(* PLC project Tc2_SUPS.FB_S_UPS_CX9020_U900 Demo, tc3-libraries-kb TwinCAT 3.1 *)
(* stored: creationDateTime 2026-05-10T09:00:00, modificationDateTime 2026-05-10T09:00:00 *)

PROGRAM P_Demo_FB_S_UPS_CX9020_U900
  VAR
    fbFB_S_UPS_CX9020_U900 : FB_S_UPS_CX9020_U900;  (* CX9020-U900 实例 *)
    arg_sNetID : T_AmsNetId;  (* VAR_INPUT sNetID: 控制器 AmsNetId（空字符串表本地） *)
    arg_iPLCPort : UINT;  (* VAR_INPUT iPLCPort: 写持久化数据的 PLC runtime 端口（851/852/...，0 = 自动） *)
    arg_tTimeout : TIME;  (* VAR_INPUT tTimeout: ADS 超时（默认 DEFAULT_ADS_TIMEOUT） *)
    arg_eUpsMode : E_S_UPS_Mode;  (* VAR_INPUT eUpsMode: UPS 工作模式（默认 eSUPS_WrPersistData_Shutdown） *)
    arg_ePersistentMode : E_PersistentMode;  (* VAR_INPUT ePersistentMode: 持久化数据写入模式（默认 SPDM_2PASS） *)
    arg_tRecoverTime : TIME;  (* VAR_INPUT tRecoverTime: 短时断电恢复时间（默认 T#10s） *)
    out_bPowerFailDetect : BOOL;  (* VAR_OUTPUT bPowerFailDetect: 断电期间为 TRUE *)
    out_eState : E_S_UPS_State;  (* VAR_OUTPUT eState: FB 内部状态 *)
  END_VAR

            // ============================================================
// Tc2_SUPS.FB_S_UPS_CX9020_U900 演示程序
// ============================================================
// 场景：在 CX9020-U900 平台上接管 1-second UPS：检测断电时保存持久数据并执行 quick shutdown
// 验证步骤：
//   1. 引用 Tc2_SUPS（及其依赖：Tc2_System 等）
//   2. 编译 + 登录
//   3. 在线监视各 out_* 输出
//   4. 必要时按场景给 arg_* 输入赋值（详见 doc.md 的'使用注意'）
// ============================================================

fbFB_S_UPS_CX9020_U900(
    sNetID := arg_sNetID,
    iPLCPort := arg_iPLCPort,
    tTimeout := arg_tTimeout,
    eUpsMode := arg_eUpsMode,
    ePersistentMode := arg_ePersistentMode,
    tRecoverTime := arg_tRecoverTime,
    bPowerFailDetect => out_bPowerFailDetect,
    eState => out_eState
);

          
END_PROGRAM
